// Mitsubishi GX Works2 project: ZhaoQing_HuaCheng2_17_12_2   PLC: Q03UDE
// 化成线2号柜

TYPE ShuttleCarIO : STRUCT
  xAuto : BOOL;  (* 自动 *)
  xManual : BOOL;  (* 手动 *)
  xReady : BOOL;  (* 准备就绪 *)
  xForward : BOOL;  (* 正转 *)
  xBackward : BOOL;  (* 反转 *)
  diCurrentPos : DINT;  (* 当前位置 *)
  diDestinationPos : DINT;  (* 目标位置 *)
  xCW : BOOL;  (* 正转输出 *)
  xCCW : BOOL;  (* 反转输出 *)
  xBrake : BOOL;  (* 刹车 *)
  xHomeSwitch : BOOL;  (* 零位接近开关 *)
  xPosLimit : BOOL;  (* 正限位 *)
  xNegLimit : BOOL;  (* 负限位 *)
  xMDIExe : BOOL;  (* MDI开始 *)
  xMDIDone : BOOL;  (* MDI 完成 *)
  xPassLimit : BOOL;  (* 限位屏蔽 *)
  xPosLimitCatch : BOOL;  (* 正限位捕捉 *)
  xNegLimitCatch : BOOL;  (* 负限位捕捉 *)
  xHomeExe : BOOL;  (* 开始寻零 *)
  xHomeDone : BOOL;  (* 寻零完成 *)
  xHomeBusy : BOOL;  (* 寻零中 *)
  xHomeFailed : BOOL;  (* 寻零失败 *)
  xBusy : BOOL;  (* 工作中 *)
  xReset : BOOL;  (* 复位 *)
END_STRUCT END_TYPE

TYPE ConveyorIO : STRUCT
  xCWPresent : BOOL;  (* 正转检测有无传感器 *)
  xCCWPresent : BOOL;  (* 反转检测有无传感器 *)
  xLoad : BOOL;  (* 上料请求 *)
  xUnload : BOOL;  (* 下料请求 *)
  xMotorCW : BOOL;  (* 电机正转 *)
  xMotorCCW : BOOL;  (* 电机反转 *)
  xEmpty : BOOL;  (* 线体状态为空 *)
  xNextRun : BOOL;  (* 下段线体运行 *)
  xLastRun : BOOL;  (* 上段线体运行 *)
  xUnloadCCW : BOOL;  (* 下料为反转 *)
  xloadCCW : BOOL;  (* 上料为反转 *)
  xLeave : BOOL;  (* 已经离开 *)
  xAuto : BOOL;  (* 自动 *)
  xManual : BOOL;  (* 手动 *)
  xForward : BOOL;  (* 正转手动 *)
  xBackward : BOOL;  (* 反转手动 *)
  strProductSerial : STRING[4];  (* 产品信息 *)
  xEStop : BOOL;  (* 急停 *)
  xReset : BOOL;  (* 复位 *)
  iProductCategory : INT;  (* 产品类型0：无料1：正极  2：负极 3：隔膜 4：空料架 *)
  xBusy : BOOL;  (* 工作中 *)
  tLeaveDelay : TIME;  (* 离开延时设置 *)
  xPutInto : BOOL;  (* 线体直接投入物料 *)
  xLoadAlarrm : BOOL;  (* 上料报警 *)
  xUnloadAlarm : BOOL;  (* 下料报警 *)
END_STRUCT END_TYPE

// global labels: Global1
VAR_GLOBAL
  g_xAuto : BOOL;
  g_xManual : BOOL;
  g_xEStop : BOOL;
  g_xReset : BOOL;
END_VAR

// task Task_01 (event TRUE, interval 0, priority 31): POU

PROGRAM POU
VAR
  H850Conveyor22 : Conveyor;
  Lifter3 : ShuttleCar;
  H850Conveyor22IO : ConveyorIO;
  H850Conveyor21 : Conveyor;
  H850Conveyor21IO : ConveyorIO;
  H850Conveyor20 : Conveyor;
  H850Conveyor20IO : ConveyorIO;
END_VAR
H850Conveyor20(ConveyorMotor:=H850Conveyor20IO);
H850Conveyor21(ConveyorMotor:=H850Conveyor21IO);
H850Conveyor22(ConveyorMotor:=H850Conveyor22IO);
H850Conveyor20IO.xAuto:=g_xAuto;
H850Conveyor20IO.xManual:=g_xManual;
H850Conveyor20IO.xForward:=M30;
H850Conveyor20IO.xCWPresent:=X8;
Y8:=H850Conveyor20IO.xMotorCW;
END_PROGRAM

FUNCTION_BLOCK ShuttleCar
VAR_IN_OUT
  ShuttleCarInOut : ShuttleCarIO;
END_VAR
VAR
  m_xBrakeDelay : BOOL;  (* 刹车延时标志位 *)
  diCurrentPosRetain : DINT;
  m_tonBrakeDelay : TON;  (* 延时 *)
  m_tBrakeDelay : TIME;
  m_xBrake : BOOL;
  m_tBrakeDelayCurrentTime : TIME;
END_VAR
(*******************************************************************
输送小车程序，可用于使用认址片控制位置的输送车程序，可用于控制提升机，
使用了限位捕捉程序防止小车惯性过大冲过限位后继续行走，捕捉程序采用反
转复位，这样设计有弊端可能反转复位后车的位置并没有回到限位以内,当两个
限位同时碰到的时候，会使运料小车进入死锁状态，通过xPassLimit来解开死锁，
可以在触摸屏中使用一个带权限的按钮来进行控制，配合ShuttleCarCurrentPos
函数来计算位置信息
修改信息  修改后请增加版本
YAO      V1.0
********************************************************************)

ShuttleCarInOut.xPosLimitCatch:=LDF(TRUE,ShuttleCarInOut.xPosLimit) OR ShuttleCarInOut.xPosLimitCatch;
IF ShuttleCarInOut.xCCW THEN  
	ShuttleCarInOut.xPosLimitCatch:=0;
END_IF;

ShuttleCarInOut.xNegLimitCatch:=LDF(TRUE,ShuttleCarInOut.xNegLimit) OR ShuttleCarInOut.xNegLimitCatch;
IF ShuttleCarInOut.xCW THEN   
	ShuttleCarInOut.xNegLimitCatch:=0;  
END_IF;
IF ShuttleCarInOut.xPassLimit OR
	(ShuttleCarInOut.xNegLimitCatch 
	AND ShuttleCarInOut.xPosLimitCatch)  THEN  
	ShuttleCarInOut.xNegLimitCatch:=0; 
	ShuttleCarInOut.xPosLimitCatch:=0;
END_IF;

IF ShuttleCarInOut.xReady THEN	
    IF ShuttleCarInOut.xManual THEN  
	    IF ShuttleCarInOut.xForward 
			AND ShuttleCarInOut.xBackward=0 
			AND ShuttleCarInOut.xCCW=0 
			AND ShuttleCarInOut.xPosLimitCatch=0 THEN
		    ShuttleCarInOut.xCW:=1;
		    ELSE
		    ShuttleCarInOut.xCW:=0;
	    END_IF;
	    IF ShuttleCarInOut.xBackward 
			AND ShuttleCarInOut.xForward=0 
			AND ShuttleCarInOut.xCW=0 
			AND ShuttleCarInOut.xNegLimitCatch=0 THEN  
		    ShuttleCarInOut.xCCW:=1;
		    ELSE
		    ShuttleCarInOut.xCCW:=0;
	    END_IF;
    END_IF;
  IF ShuttleCarInOut.xAuto THEN  
	  IF ShuttleCarInOut.xMDIExe AND ShuttleCarInOut.diDestinationPos<>0 THEN
	
	    IF ShuttleCarInOut.diCurrentPos<ShuttleCarInOut.diDestinationPos AND ShuttleCarInOut.xPosLimitCatch=0 THEN
			ShuttleCarInOut.xCW:=1;
			ShuttleCarInOut.xCCW:=0;
			ShuttleCarInOut.xMDIDone:=0;
		END_IF;

		IF ShuttleCarInOut.diCurrentPos>ShuttleCarInOut.diDestinationPos AND ShuttleCarInOut.xNegLimitCatch=0 THEN
			ShuttleCarInOut.xCCW:=1;
			ShuttleCarInOut.xCW:=0;
			ShuttleCarInOut.xMDIDone:=0;
		END_IF;
	
		IF ShuttleCarInOut.diCurrentPos=ShuttleCarInOut.diDestinationPos THEN
			ShuttleCarInOut.xCW:=0;
			ShuttleCarInOut.xCCW:=0;
			ShuttleCarInOut.xMDIDone:=1;
			ELSE
			ShuttleCarInOut.xMDIDone:=0;
		END_IF;

		IF ShuttleCarInOut.xPosLimitCatch THEN
			ShuttleCarInOut.xCW:=0;
			ShuttleCarInOut.xMDIDone:=0;
		END_IF;

		IF ShuttleCarInOut.xNegLimitCatch THEN
			ShuttleCarInOut.xCCW:=0;
			ShuttleCarInOut.xMDIDone:=0;
		END_IF;
		ELSE
		ShuttleCarInOut.xCW:=0;
		ShuttleCarInOut.xCCW:=0;
		ShuttleCarInOut.xMDIDone:=0;
	  END_IF;
	END_IF;
END_IF;

m_tonBrakeDelay(IN:=m_xBrakeDelay ,PT:= T#40MS,Q:=m_xBrake ,ET:= m_tBrakeDelayCurrentTime);
IF (ShuttleCarInOut.xCW OR ShuttleCarInOut.xCCW) AND ShuttleCarInOut.xReady=1 THEN
	ShuttleCarInOut.xBrake:=m_xBrake;
	m_xBrakeDelay:=1;
	ELSE
	ShuttleCarInOut.xBrake:=0;
	m_xBrakeDelay:=0;
END_IF;

IF SM402 THEN 
	ShuttleCarInOut.diCurrentPos:=diCurrentPosRetain;
	ELSE
	diCurrentPosRetain:=ShuttleCarInOut.diCurrentPos;
END_IF;

IF ShuttleCarInOut.xCW OR ShuttleCarInOut.xCCW THEN
	ShuttleCarInOut.xBusy:=1;
	ELSE
	ShuttleCarInout.xBusy:=0;
END_IF;
END_FUNCTION_BLOCK

FUNCTION_BLOCK Conveyor
VAR
  tRundelay : TIME;  (* 离开延时 *)
END_VAR
VAR_IN_OUT
  ConveyorMotor : ConveyorIO;  (* 输送线输入输出 *)
END_VAR
VAR
  iStep : INT;  (* 上料步骤 *)
  m_tLoadTimer : TIME;  (* 上料计时器 *)
  m_tUnloadTimer : TIME;  (* 下料计时器 *)
  m_tonLeaveDelay : TON;  (* 离开延时定时器 *)
  m_xLeaveDelayOut : BOOL;  (* 离开延时 *)
  m_tLeaveCurrentTime : TIME;
  m_tonLoadAlarm : TON;  (* 上料延时报警 *)
END_VAR
VAR CONSTANT
  LOAD_UNLOAD_TIME : TIME := T#30s;  (* 延时报警常量 *)
END_VAR
VAR
  m_tonUnloadAlam : TON;  (* 下料报警定时器 *)
END_VAR
(*////////////////////////////////////////////////////////////////////////////////////////////////////////////
//传输线控制FB块，可控制单方向线体，双向旋转线体，支持双向上下料            
//线体初始化后为空的情况下输入xLoad信号即可进行上料动作，使用xLoadCCW信号可反方向上料
//增加了产品信息和产品种类的储存，当传输线为空和上料进行标志位为零的情况下清除产品信息和产品种类
//使用方式是在置位xLoad信号后，把产品信息和产品种类传入，等下料后自动清零
//线体不为空的情况下使用xUnload信号可进行下料动作，物料有无传感器的下降沿后出发计时器，延时断开传输线旋转
//单方向传输线体把xLoadCCW、xUnloadCCW设置为零，双向线体上料方向和下料反向的,方向固定的 把xUnloadCCW设置为1
//双方向线体双向都能上下料的要根据上料的方向来设置xLoadCCW,xUnloadCCW
//增加工作中信号xBusy当电机正转 显示为工作中
//增加上下料超时报警，xLoadAlarm，xUnloadAlarm，设定时间在LOAD_UNLOAD_TIME常量上，现在设置的为30秒
//增加xPutInto信号，用于直接投入的物料，检测开关感应到后，直接进入下料流程，上升沿有效
//离开延时改为变量 iLeaveDelay 默认为0 离开检测开关离输送线尾端比较远的线体需要根据情况设定100ms为单位
//修改信息  修改后请增加版本
//YAO      V1.0
///////////////////////////////////////////////////////////////////////////////////////////////////////////
********************************************************)


IF ConveyorMotor.xAuto THEN
CASE iStep OF
	0:
	ConveyorMotor.xMotorCW:=0;
	ConveyorMotor.xMotorCCW:=0;
	ConveyorMotor.xNextRun:=0;

	IF (ConveyorMotor.xCWPresent OR ConveyorMotor.xCCWPresent) 
		AND ConveyorMotor.xEStop=0 
		AND ConveyorMotor.xLoadAlarrm = 0
		AND ConveyorMotor.xUnloadAlarm = 0 THEN
		iStep:=3;
		ConveyorMotor.xEmpty:=0;
		ELSE
		iStep:=1;
		ConveyorMotor.xEmpty:=1;
	END_IF;
		
	1: 
	IF ConveyorMotor.xLoad    
		AND ConveyorMotor.xMotorCW=0   
		AND ConveyorMotor.xMotorCCW=0   
		AND ConveyorMotor.xEmpty THEN	
		iStep:=2;
	END_IF;
	2: 
	IF ConveyorMotor.xloadCCW THEN
		ConveyorMotor.xMotorCCW:=1; 
		ConveyorMotor.xMotorCW:=0;
		IF ConveyorMotor.xCCWPresent THEN
			iStep:=3;
		END_IF;
		ELSE
	    ConveyorMotor.xMotorCW:=1;  
		ConveyorMotor.xMotorCCW:=0;
	    IF ConveyorMotor.xCWPresent THEN 	 
		    iStep:=3;
		END_IF;
	END_IF;
	3:
	ConveyorMotor.xMotorCW:=0;
	ConveyorMotor.xMotorCCW:=0;
	ConveyorMotor.xEmpty:=0;
	IF ConveyorMotor.xUnload THEN 
		iStep:=4;
	END_IF;
	4:	
	IF ConveyorMotor.xUnloadCCW THEN   
		ConveyorMotor.xMotorCCW:=1;  
		ConveyorMotor.xMotorCW:=0;

		ConveyorMotor.xLeave:=ldf(TRUE,ConveyorMotor.xCCWPresent) OR ConveyorMotor.xLeave;
		ELSE
	    ConveyorMotor.xMotorCW:=1;  
		ConveyorMotor.xMotorCCW:=0;
		ConveyorMotor.xLeave:=ldf(TRUE,ConveyorMotor.xCWPresent) OR ConveyorMotor.xLeave;
	END_IF;
	ConveyorMotor.xNextRun:=1; 
	m_tonLeaveDelay(IN:= ConveyorMotor.xLeave,PT:= ConveyorMotor.tLeaveDelay,Q:=m_xLeaveDelayOut ,ET:= m_tLeaveCurrentTime );	
	IF m_xLeaveDelayOut THEN
		ConveyorMotor.xMotorCW:=0;
		ConveyorMotor.xMotorCCW:=0;
		iStep:=0;
		ConveyorMotor.xNextRun:=0;
		ConveyorMotor.xLeave:=0;
		ConveyorMotor.xEmpty:=1;		
	END_IF;	
	IF NOT ConveyorMotor.xUnload THEN 
		istep:=0;
	END_IF;
END_CASE;
IF LDP(TRUE,ConveyorMotor.xPutInto) THEN
	iStep:=0;
END_IF;
END_IF;
IF ConveyorMotor.xEmpty AND NOT ConveyorMotor.xLoad THEN
	ConveyorMotor.strProductSerial:='';
	ConveyorMotor.iProductCategory:=0;
END_IF;
IF ConveyorMotor.xEStop OR ConveyorMotor.xReset THEN
	iStep:=0;
END_IF;	

IF ConveyorMotor.xManual THEN
	iStep:=0;

	IF ConveyorMotor.xForward 
		AND ConveyorMotor.xBackward=0 
		AND ConveyorMotor.xMotorCCW=0 THEN
		ConveyorMotor.xMotorCW:=1;
		ConveyorMotor.xMotorCCW:=0;
		ELSE
		ConveyorMotor.xMotorCW:=0;
	END_IF;

	IF ConveyorMotor.xBackward 
		AND ConveyorMotor.xForward=0 
		AND ConveyorMotor.xMotorCW=0  THEN
		ConveyorMotor.xMotorCCW:=1;
		conveyormotor.xMotorCW:=0;
		ELSE
		ConveyorMotor.xMotorCCW:=0;
	END_IF;
END_IF;
IF ConveyorMotor.xMotorCCW        
	OR ConveyorMotor.xMotorCW THEN  
	ConveyorMotor.xBusy:=1;
	ELSE
	ConveyorMotor.xBusy:=0;
END_IF;
m_tonLoadAlarm(IN:= iStep=2 ,PT:= LOAD_UNLOAD_TIME,Q:= ConveyorMotor.xLoadAlarrm ,ET:= m_tLoadTimer );
m_tonUnloadAlam(IN:= iStep=4,PT:= LOAD_UNLOAD_TIME,Q:= ConveyorMotor.xUnloadAlarm,ET:= m_tUnloadTimer );
(*OUT_T(iStep=2,m_tLoadTimer,LOAD_UNLOAD_TIME);
OUT_T(iStep=4,m_tUnloadTimer,LOAD_UNLOAD_TIME);
ConveyorMotor.xLoadAlarrm:=m_tLoadTimer.S;
ConveyorMotor.xUnloadAlarm:=m_tUnloadTimer.S;*)
END_FUNCTION_BLOCK
